TYPE (* Typedef of the ISO CF/user information data array *)
  (* Version 1.0, 2025-09-04, Franz Höpfinger, initial API and implementation and/or initial documentation *)
  PACKAGE isobus::pgn;
  CF_NAME_T : STRUCT
    data : ARRAY [0..7] OF BYTE := [16#FF, 16#FF, 16#FF, 16#FF, 16#FF, 16#FF, 16#FF, 16#FF];
  END_STRUCT;
END_TYPE
